FUNCTION_BLOCK RobotPPScheduler
VAR
	/// Interfaces
	_robot_interface_adr: POINTER TO RobotInterface;
	_motor_pp_scheduler_adr: POINTER TO ARRAY[0..1] OF MotorPPScheduler;
END_VAR
VAR
	/// Runtime variables
	_robot_state : robot_pp_states_t:=robot_pp_states_t.END;
	_target_distance: LREAL;
	_target_angle : LREAL;
	_motor_angles : ARRAY[0..1] OF DINT;
END_VAR

IF(_robot_interface_adr^.robot_mode=robot_modes_t.PP  AND _robot_interface_adr^.robot_enabled) THEN
	CASE _robot_state OF
		robot_pp_states_t.START:
			_motor_pp_scheduler_adr^[0].activate();
			_motor_pp_scheduler_adr^[1].activate();
			InverseKinematics(	target_dist:=_target_distance, 
								target_angle:=_target_angle,
								motor_axis1_angle=>_motor_angles[0],
								motor_axis2_angle=>_motor_angles[1]);
			_motor_pp_scheduler_adr^[0].start_operation(
									target_position:=_motor_angles[0],
									change_immediately:=TRUE,
									reference_coordinate:=FALSE,
									push_operation:=FALSE);
			_motor_pp_scheduler_adr^[1].start_operation(
									target_position:=_motor_angles[1],
									change_immediately:=TRUE,
									reference_coordinate:=FALSE,
									push_operation:=FALSE);
			_robot_state:=robot_pp_states_t.INPROGRESS;
		robot_pp_states_t.INPROGRESS:
			IF(_motor_pp_scheduler_adr^[0].get_state()=motor_pp_states_t.END AND _motor_pp_scheduler_adr^[1].get_state()=motor_pp_states_t.END) THEN
				_robot_state:=robot_pp_states_t.END;
			END_IF
	END_CASE
END_IF

{attribute 'TcRpcEnable'}
METHOD activate : BOOL
VAR_INPUT
END_VAR

_robot_interface_adr^.robot_mode:=robot_modes_t.PP;
_robot_state:=robot_pp_states_t.END;
END_METHOD

METHOD FB_init : BOOL
VAR_INPUT
	bInitRetains : BOOL; // if TRUE, the retain variables are initialized (warm start / cold start)
	bInCopyCode : BOOL;  // if TRUE, the instance afterwards gets moved into the copy code (online change)
	robot_interface_adr: POINTER TO RobotInterface;
END_VAR
_robot_interface_adr:=robot_interface_adr;
_motor_pp_scheduler_adr:=_robot_interface_adr^.motor_pp_scheduler_adr;
END_METHOD

{attribute 'TcRpcEnable'}
METHOD get_state : robot_pp_states_t
VAR_INPUT
END_VAR
get_state:=_robot_state;
END_METHOD

{attribute 'TcRpcEnable'}
METHOD start_operation : BOOL
VAR_INPUT
	target_distance: LREAL;
	target_angle : LREAL;
END_VAR
_robot_interface_adr^.robot_enabled:=TRUE;
_target_distance:=target_distance;
_target_angle:=target_angle;
_robot_state:=robot_pp_states_t.START;
END_METHOD

END_FUNCTION_BLOCK

(* stored: Version 1.1.0.1, ProductVersion 3.1.4024.12
   POU RobotPPScheduler: Id {9b32e0d7-ad1e-41c9-a248-d2e0e521ae2c}, SpecialFunc None
   Method activate: Id {1f76cf63-a8c1-4183-aed0-d741a94f6c79}
   Method FB_init: Id {6e97cf44-629f-4b76-895c-5ab90765f727}
   Method get_state: Id {69a9beaa-8d00-4706-8acd-3d775c010d33}
   Method start_operation: Id {febac2b4-e500-4d4d-bee1-3bfd170097fa} *)
